// SIMATIC STEP 7 (V5.x) project TEMA 13 EJERCICIO 41
// CPU: CPU313 C-2 DP(1)
// station: P_ADR_BUS
// station: Hardware
// station: Equipo SIMATIC 300
// program: Programa S7(1)

SYMBOL_TABLE
"FLANCOS"	DB 1	DB 1
"MANIOBRA"	DB 2	DB 2
"P MARCHA"	I 0.0	BOOL
"P PARO"	I 0.1	BOOL
"P CAMBIO DE SENTIDO"	I 0.2	BOOL
"Cycle Execution"	OB 1	OB 1
"M1 LINEA"	Q 0.0	BOOL
"M1ESTRELLA"	Q 0.1	BOOL
"M1 TRIANGULO"	Q 0.2	BOOL
"CINTA 1"	Q 0.3	BOOL
"CINTA 2 IZQUIERDAS"	Q 0.4	BOOL
"CINTA 2 DERECHAS"	Q 0.5	BOOL
END_SYMBOL_TABLE

DATA_BLOCK "FLANCOS"	// DB 1
VERSION : 0.1
  STRUCT
   M0 : BOOL ;
   M1 : BOOL ;
   M2 : BOOL ;
   M3 : BOOL ;
   M4 : BOOL ;
   M5 : BOOL ;
   M6 : BOOL ;
   M7 : BOOL ;
   M10 : BOOL ;
   M11 : BOOL ;
   M12 : BOOL ;
   M13 : BOOL ;
   M14 : BOOL ;
   M15 : BOOL ;
   M16 : BOOL ;
   M17 : BOOL ;
   M20 : BOOL ;
   M21 : BOOL ;
   M22 : BOOL ;
   M23 : BOOL ;
  END_STRUCT ;	
BEGIN
END_DATA_BLOCK

DATA_BLOCK "MANIOBRA"	// DB 2
VERSION : 0.1
  STRUCT
   M0 : BOOL ;
   M1 : BOOL ;
   M2 : BOOL ;
   M3 : BOOL ;
   M4 : BOOL ;
   M5 : BOOL ;
   M6 : BOOL ;
   M7 : BOOL ;
  END_STRUCT ;	
BEGIN
END_DATA_BLOCK

ORGANIZATION_BLOCK "Cycle Execution"	// OB 1
TITLE = "Main Program Sweep (Cycle)"
VERSION : 0.1
VAR_TEMP
  OB1_EV_CLASS : BYTE ;	//Bits 0-3 = 1 (Coming event), Bits 4-7 = 1 (Event class 1)
  OB1_SCAN_1 : BYTE ;	//1 (Cold restart scan 1 of OB 1), 3 (Scan 2-n of OB 1)
  OB1_PRIORITY : BYTE ;	//Priority of OB Execution
  OB1_OB_NUMBR : BYTE ;	//1 (Organization block 1, OB1)
  OB1_RESERVED_1 : BYTE ;	//Reserved for system
  OB1_RESERVED_2 : BYTE ;	//Reserved for system
  OB1_PREV_CYCLE : INT ;	//Cycle time of previous OB1 scan (milliseconds)
  OB1_MIN_CYCLE : INT ;	//Minimum cycle time of OB1 (milliseconds)
  OB1_MAX_CYCLE : INT ;	//Maximum cycle time of OB1 (milliseconds)
  OB1_DATE_TIME : DATE_AND_TIME ;	//Date and time OB1 started
END_VAR
BEGIN
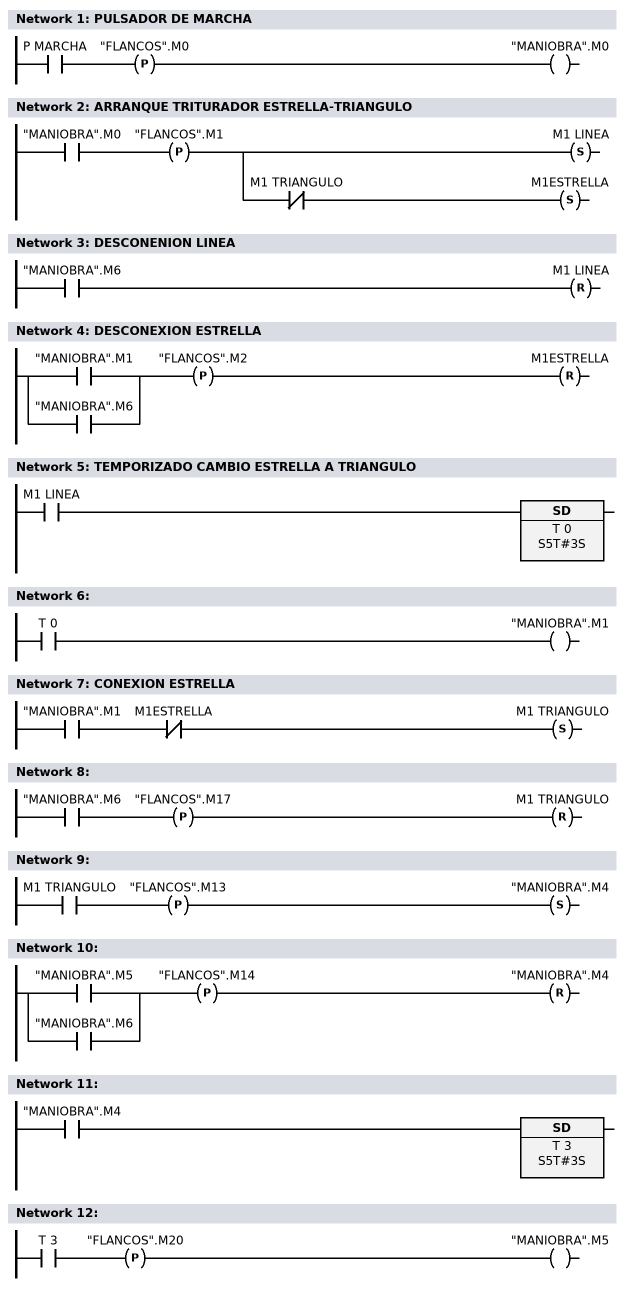
NETWORK
TITLE = PULSADOR DE MARCHA
      A     "P MARCHA";
      FP    "FLANCOS".M0;
      =     "MANIOBRA".M0;
NETWORK
TITLE = ARRANQUE TRITURADOR ESTRELLA-TRIANGULO
//EN PRIMER LUGAR CONNECTA LINEA Y ESTRELLA
      A     "MANIOBRA".M0;
      FP    "FLANCOS".M1;
      =     L 20.0;
      A     L 20.0;
      BLD   102;
      S     "M1 LINEA";
      A     L 20.0;
      AN    "M1 TRIANGULO";
      S     "M1ESTRELLA";
NETWORK
TITLE = DESCONENION LINEA
      A     "MANIOBRA".M6;
      R     "M1 LINEA";
NETWORK
TITLE = DESCONEXION ESTRELLA
      A(;
      O     "MANIOBRA".M1;
      O     "MANIOBRA".M6;
      );
      FP    "FLANCOS".M2;
      R     "M1ESTRELLA";
NETWORK
TITLE = TEMPORIZADO CAMBIO ESTRELLA A TRIANGULO
      A     "M1 LINEA";
      L     S5T#3S;
      SD    T 0;
NETWORK
TITLE =
      A     T 0;
      =     "MANIOBRA".M1;
NETWORK
TITLE = CONEXION ESTRELLA
      A     "MANIOBRA".M1;
      AN    "M1ESTRELLA";
      S     "M1 TRIANGULO";
NETWORK
TITLE =
      A     "MANIOBRA".M6;
      FP    "FLANCOS".M17;
      R     "M1 TRIANGULO";
NETWORK
TITLE =
      A     "M1 TRIANGULO";
      FP    "FLANCOS".M13;
      S     "MANIOBRA".M4;
NETWORK
TITLE =
      A(;
      O     "MANIOBRA".M5;
      O     "MANIOBRA".M6;
      );
      FP    "FLANCOS".M14;
      R     "MANIOBRA".M4;
NETWORK
TITLE =
      A     "MANIOBRA".M4;
      L     S5T#3S;
      SD    T 3;
NETWORK
TITLE =
      A     T 3;
      FP    "FLANCOS".M20;
      =     "MANIOBRA".M5;
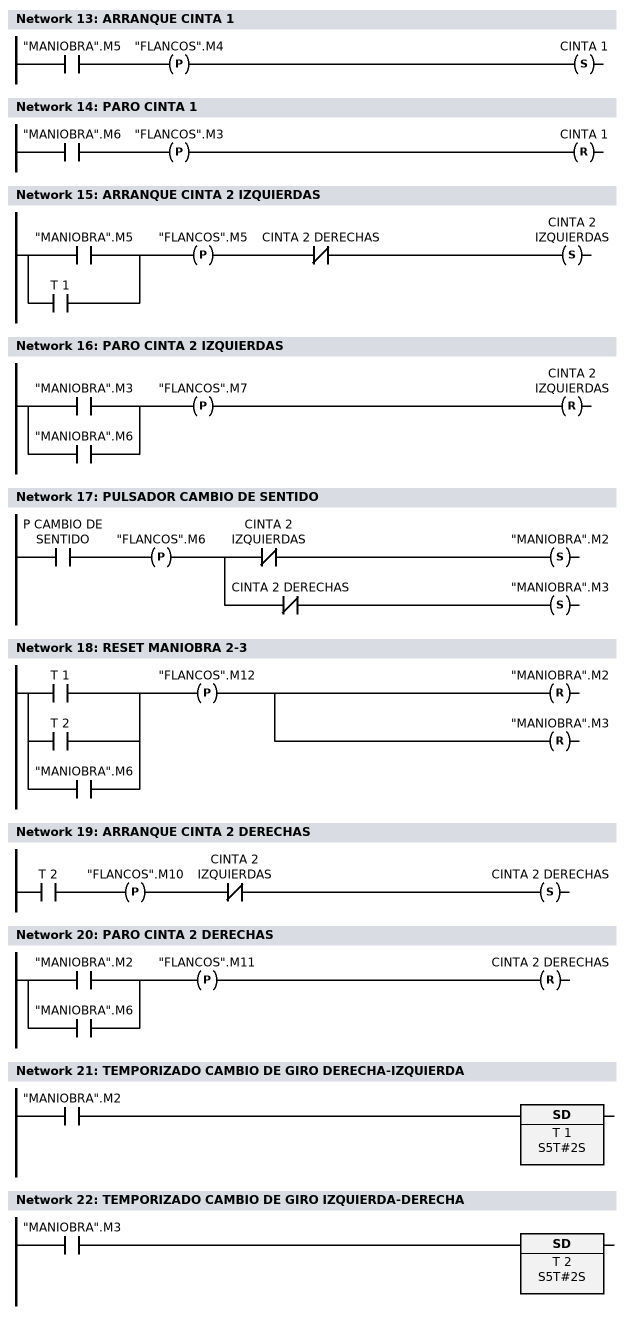
NETWORK
TITLE = ARRANQUE CINTA 1 
      A     "MANIOBRA".M5;
      FP    "FLANCOS".M4;
      S     "CINTA 1";
NETWORK
TITLE = PARO CINTA 1 
      A     "MANIOBRA".M6;
      FP    "FLANCOS".M3;
      R     "CINTA 1";
NETWORK
TITLE = ARRANQUE CINTA 2 IZQUIERDAS
      A(;
      O     "MANIOBRA".M5;
      O     T 1;
      );
      FP    "FLANCOS".M5;
      AN    "CINTA 2 DERECHAS";
      S     "CINTA 2 IZQUIERDAS";
NETWORK
TITLE = PARO CINTA 2 IZQUIERDAS
      A(;
      O     "MANIOBRA".M3;
      O     "MANIOBRA".M6;
      );
      FP    "FLANCOS".M7;
      R     "CINTA 2 IZQUIERDAS";
NETWORK
TITLE = PULSADOR CAMBIO DE SENTIDO
      A     "P CAMBIO DE SENTIDO";
      FP    "FLANCOS".M6;
      =     L 20.0;
      A     L 20.0;
      AN    "CINTA 2 IZQUIERDAS";
      S     "MANIOBRA".M2;
      A     L 20.0;
      AN    "CINTA 2 DERECHAS";
      S     "MANIOBRA".M3;
NETWORK
TITLE = RESET MANIOBRA 2-3
      A(;
      O     T 1;
      O     T 2;
      O     "MANIOBRA".M6;
      );
      FP    "FLANCOS".M12;
      R     "MANIOBRA".M2;
      R     "MANIOBRA".M3;
NETWORK
TITLE = ARRANQUE CINTA 2 DERECHAS
      A     T 2;
      FP    "FLANCOS".M10;
      AN    "CINTA 2 IZQUIERDAS";
      S     "CINTA 2 DERECHAS";
NETWORK
TITLE = PARO CINTA 2 DERECHAS
      A(;
      O     "MANIOBRA".M2;
      O     "MANIOBRA".M6;
      );
      FP    "FLANCOS".M11;
      R     "CINTA 2 DERECHAS";
NETWORK
TITLE = TEMPORIZADO CAMBIO DE GIRO DERECHA-IZQUIERDA
      A     "MANIOBRA".M2;
      L     S5T#2S;
      SD    T 1;
NETWORK
TITLE = TEMPORIZADO CAMBIO DE GIRO IZQUIERDA-DERECHA
      A     "MANIOBRA".M3;
      L     S5T#2S;
      SD    T 2;
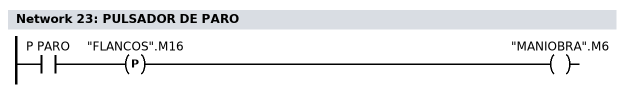
NETWORK
TITLE = PULSADOR DE PARO
      A     "P PARO";
      FP    "FLANCOS".M16;
      =     "MANIOBRA".M6;
END_ORGANIZATION_BLOCK
